// Mitsubishi GX Works2 project: test1   PLC: Q03UDV

PROGRAM MAIN
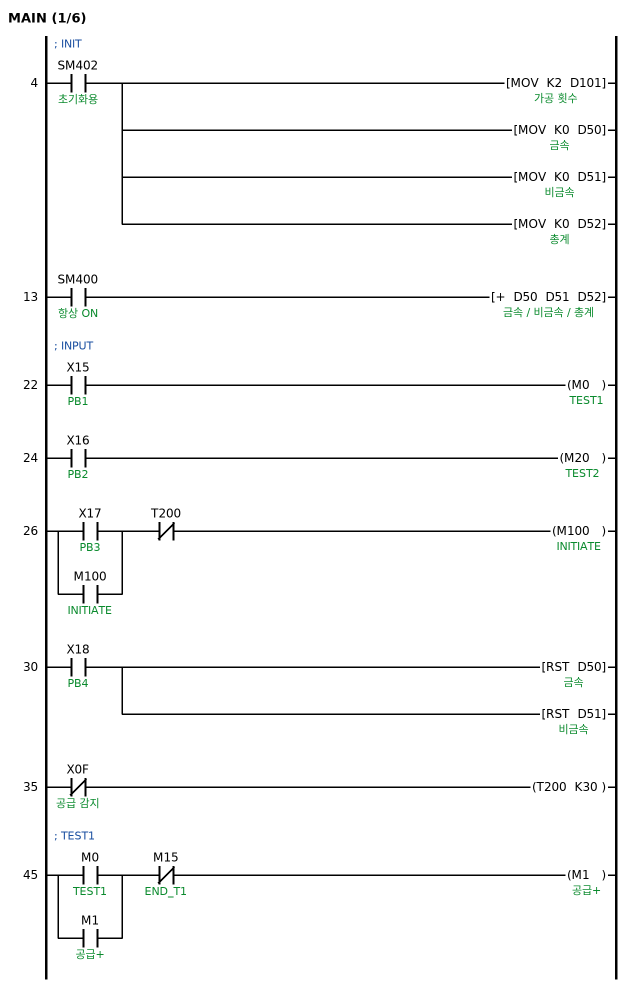
; INIT
4     LD      SM402  ; 초기화용
      MOV     K2 D101  ; 가공 횟수
      MOV     K0 D50  ; 금속
      MOV     K0 D51  ; 비금속
      MOV     K0 D52  ; 총계
13    LD      SM400  ; 항상 ON
      +       D50 D51 D52
; INPUT
22    LD      X15  ; PB1
      OUT     M0  ; TEST1
24    LD      X16  ; PB2
      OUT     M20  ; TEST2
26    LD      X17  ; PB3
      OR      M100  ; INITIATE
      ANI     T200
      OUT     M100  ; INITIATE
30    LD      X18  ; PB4
      RST     D50  ; 금속
      RST     D51  ; 비금속
35    LDI     X0F  ; 공급 감지
      OUT     T200 K30
; TEST1
45    LD      M0  ; TEST1
      OR      M1  ; 공급+
      ANI     M15  ; END_T1
      OUT     M1  ; 공급+
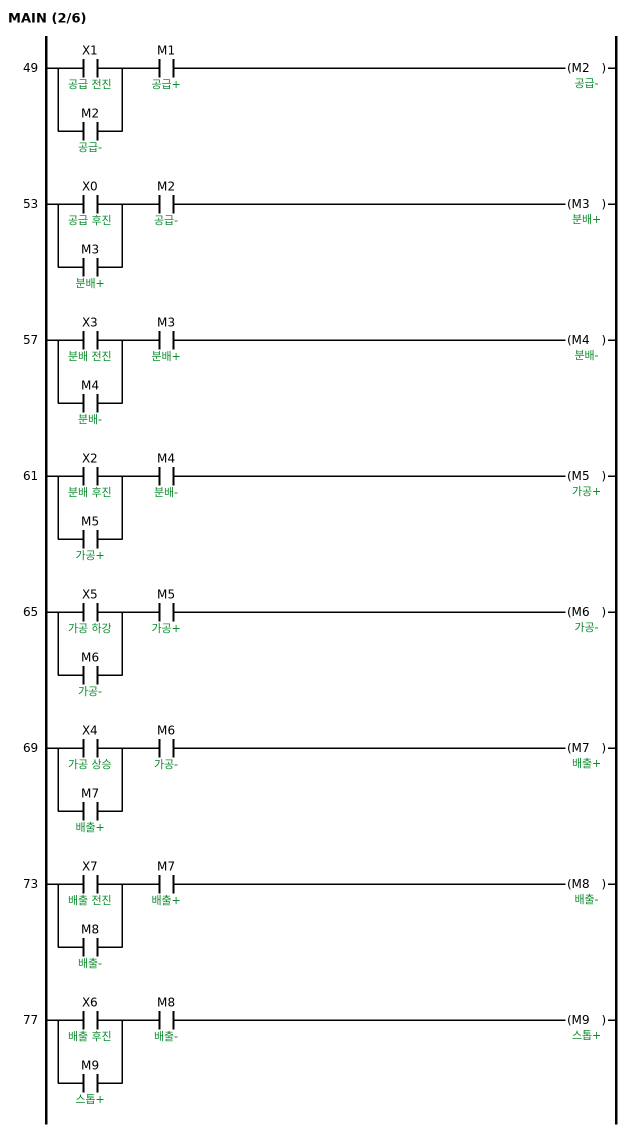
49    LD      X1  ; 공급 전진
      OR      M2  ; 공급-
      AND     M1  ; 공급+
      OUT     M2  ; 공급-
53    LD      X0  ; 공급 후진
      OR      M3  ; 분배+
      AND     M2  ; 공급-
      OUT     M3  ; 분배+
57    LD      X3  ; 분배 전진
      OR      M4  ; 분배-
      AND     M3  ; 분배+
      OUT     M4  ; 분배-
61    LD      X2  ; 분배 후진
      OR      M5  ; 가공+
      AND     M4  ; 분배-
      OUT     M5  ; 가공+
65    LD      X5  ; 가공 하강
      OR      M6  ; 가공-
      AND     M5  ; 가공+
      OUT     M6  ; 가공-
69    LD      X4  ; 가공 상승
      OR      M7  ; 배출+
      AND     M6  ; 가공-
      OUT     M7  ; 배출+
73    LD      X7  ; 배출 전진
      OR      M8  ; 배출-
      AND     M7  ; 배출+
      OUT     M8  ; 배출-
77    LD      X6  ; 배출 후진
      OR      M9  ; 스톱+
      AND     M8  ; 배출-
      OUT     M9  ; 스톱+
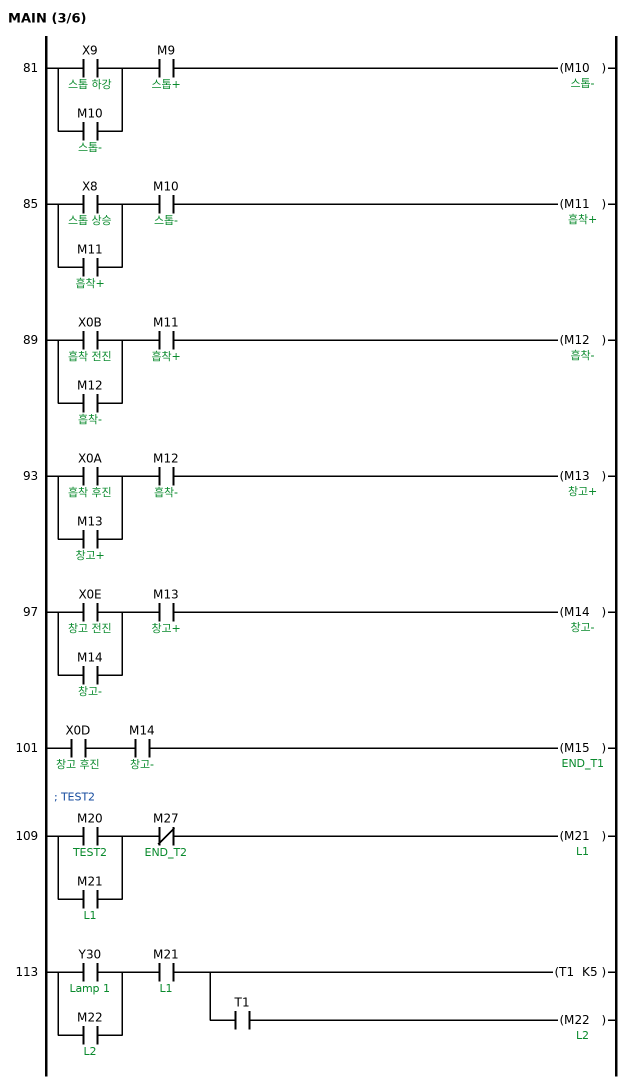
81    LD      X9  ; 스톱 하강
      OR      M10  ; 스톱-
      AND     M9  ; 스톱+
      OUT     M10  ; 스톱-
85    LD      X8  ; 스톱 상승
      OR      M11  ; 흡착+
      AND     M10  ; 스톱-
      OUT     M11  ; 흡착+
89    LD      X0B  ; 흡착 전진
      OR      M12  ; 흡착-
      AND     M11  ; 흡착+
      OUT     M12  ; 흡착-
93    LD      X0A  ; 흡착 후진
      OR      M13  ; 창고+
      AND     M12  ; 흡착-
      OUT     M13  ; 창고+
97    LD      X0E  ; 창고 전진
      OR      M14  ; 창고-
      AND     M13  ; 창고+
      OUT     M14  ; 창고-
101   LD      X0D  ; 창고 후진
      AND     M14  ; 창고-
      OUT     M15  ; END_T1
; TEST2
109   LD      M20  ; TEST2
      OR      M21  ; L1
      ANI     M27  ; END_T2
      OUT     M21  ; L1
113   LD      Y30  ; Lamp 1
      OR      M22  ; L2
      AND     M21  ; L1
      OUT     T1 K5
      AND     T1
      OUT     M22  ; L2
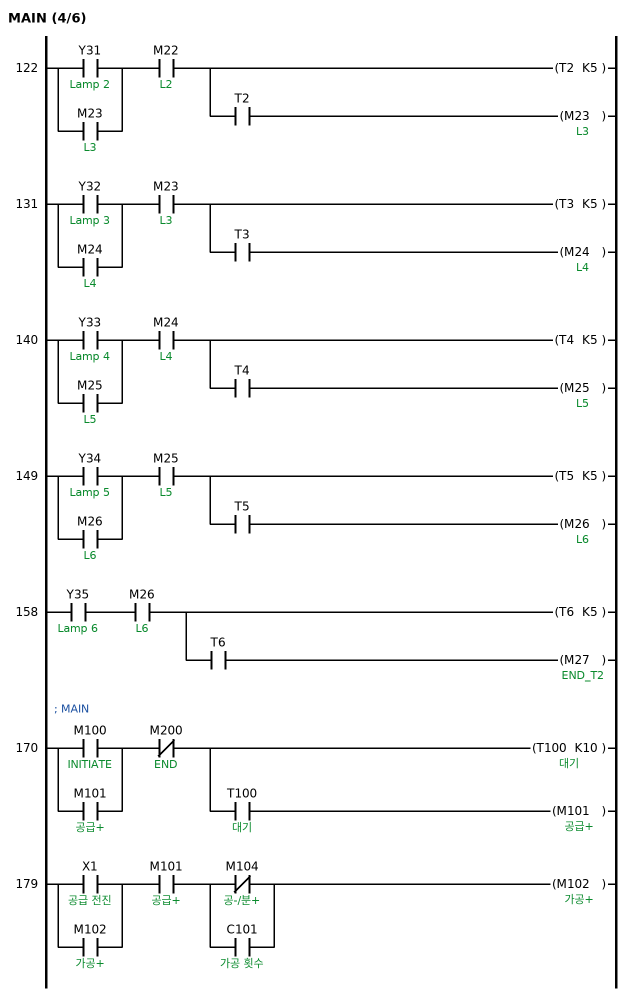
122   LD      Y31  ; Lamp 2
      OR      M23  ; L3
      AND     M22  ; L2
      OUT     T2 K5
      AND     T2
      OUT     M23  ; L3
131   LD      Y32  ; Lamp 3
      OR      M24  ; L4
      AND     M23  ; L3
      OUT     T3 K5
      AND     T3
      OUT     M24  ; L4
140   LD      Y33  ; Lamp 4
      OR      M25  ; L5
      AND     M24  ; L4
      OUT     T4 K5
      AND     T4
      OUT     M25  ; L5
149   LD      Y34  ; Lamp 5
      OR      M26  ; L6
      AND     M25  ; L5
      OUT     T5 K5
      AND     T5
      OUT     M26  ; L6
158   LD      Y35  ; Lamp 6
      AND     M26  ; L6
      OUT     T6 K5
      AND     T6
      OUT     M27  ; END_T2
; MAIN
170   LD      M100  ; INITIATE
      OR      M101  ; 공급+
      ANI     M200  ; END
      OUT     T100 K10  ; 대기
      AND     T100  ; 대기
      OUT     M101  ; 공급+
179   LD      X1  ; 공급 전진
      OR      M102  ; 가공+
      AND     M101  ; 공급+
      LDI     M104  ; 공-/분+
      OR      C101  ; 가공 횟수
      ANB
      OUT     M102  ; 가공+
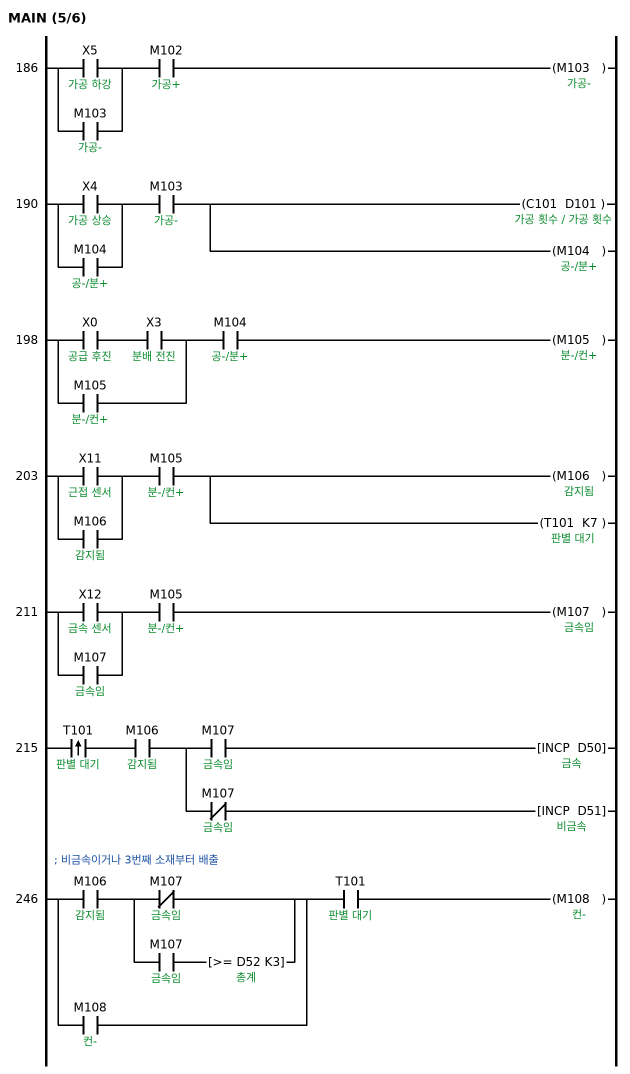
186   LD      X5  ; 가공 하강
      OR      M103  ; 가공-
      AND     M102  ; 가공+
      OUT     M103  ; 가공-
190   LD      X4  ; 가공 상승
      OR      M104  ; 공-/분+
      AND     M103  ; 가공-
      OUT     C101 D101  ; 가공 횟수 / 가공 횟수
      OUT     M104  ; 공-/분+
198   LD      X0  ; 공급 후진
      AND     X3  ; 분배 전진
      OR      M105  ; 분-/컨+
      AND     M104  ; 공-/분+
      OUT     M105  ; 분-/컨+
203   LD      X11  ; 근접 센서
      OR      M106  ; 감지됨
      AND     M105  ; 분-/컨+
      OUT     M106  ; 감지됨
      OUT     T101 K7  ; 판별 대기
211   LD      X12  ; 금속 센서
      OR      M107  ; 금속임
      AND     M105  ; 분-/컨+
      OUT     M107  ; 금속임
215   LDP     T101  ; 판별 대기
      AND     M106  ; 감지됨
      MPS
      AND     M107  ; 금속임
      INCP    D50
      MPP
      ANI     M107  ; 금속임
      INCP    D51
; 비금속이거나 3번째 소재부터 배출
246   LD      M106  ; 감지됨
      LDI     M107  ; 금속임
      LD      M107  ; 금속임
      AND>=   D52 K3  ; 총계
      ORB
      ANB
      OR      M108  ; 컨-
      AND     T101  ; 판별 대기
      OUT     M108  ; 컨-
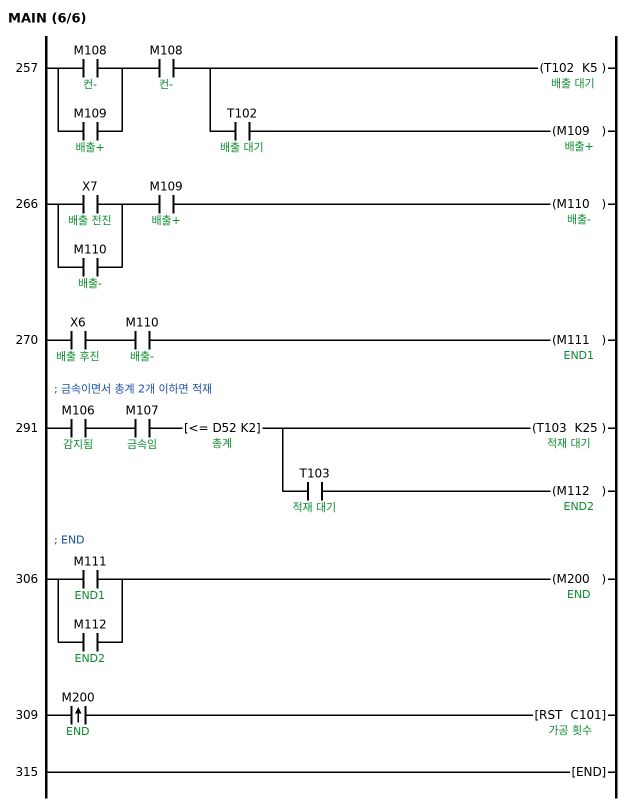
257   LD      M108  ; 컨-
      OR      M109  ; 배출+
      AND     M108  ; 컨-
      OUT     T102 K5  ; 배출 대기
      AND     T102  ; 배출 대기
      OUT     M109  ; 배출+
266   LD      X7  ; 배출 전진
      OR      M110  ; 배출-
      AND     M109  ; 배출+
      OUT     M110  ; 배출-
270   LD      X6  ; 배출 후진
      AND     M110  ; 배출-
      OUT     M111  ; END1
; 금속이면서 총계 2개 이하면 적재
291   LD      M106  ; 감지됨
      AND     M107  ; 금속임
      AND<=   D52 K2  ; 총계
      OUT     T103 K25  ; 적재 대기
      AND     T103  ; 적재 대기
      OUT     M112  ; END2
; END
306   LD      M111  ; END1
      OR      M112  ; END2
      OUT     M200  ; END
309   LDP     M200  ; END
      RST     C101  ; 가공 횟수
315   END
END_PROGRAM

PROGRAM OUTPUT
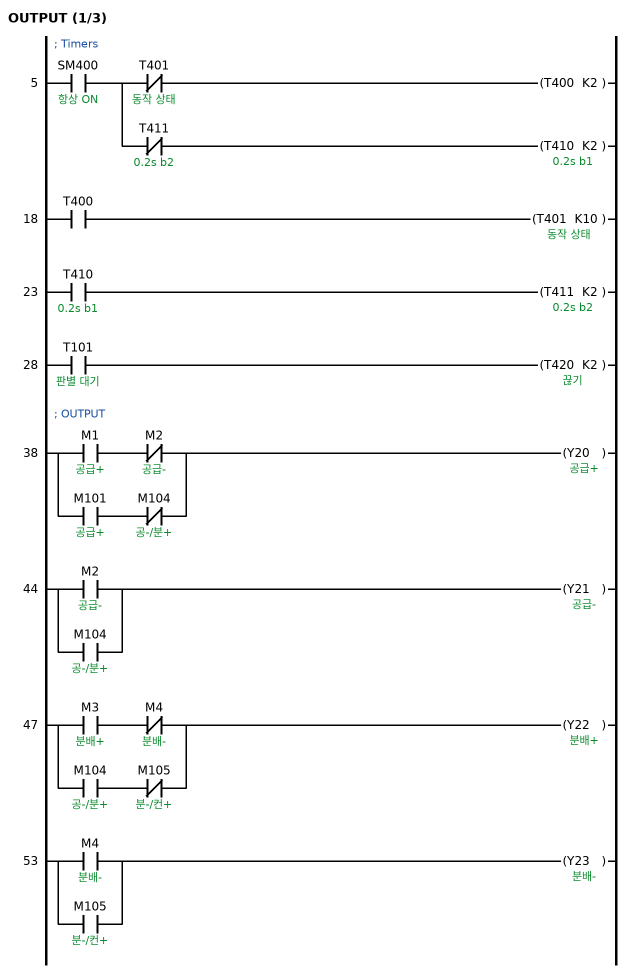
; Timers
5     LD      SM400  ; 항상 ON
      MPS
      ANI     T401  ; 동작 상태
      OUT     T400 K2
      MPP
      ANI     T411  ; 0.2s b2
      OUT     T410 K2  ; 0.2s b1
18    LD      T400
      OUT     T401 K10  ; 동작 상태
23    LD      T410  ; 0.2s b1
      OUT     T411 K2  ; 0.2s b2
28    LD      T101  ; 판별 대기
      OUT     T420 K2  ; 끊기
; OUTPUT
38    LD      M1  ; 공급+
      ANI     M2  ; 공급-
      LD      M101  ; 공급+
      ANI     M104  ; 공-/분+
      ORB
      OUT     Y20  ; 공급+
44    LD      M2  ; 공급-
      OR      M104  ; 공-/분+
      OUT     Y21  ; 공급-
47    LD      M3  ; 분배+
      ANI     M4  ; 분배-
      LD      M104  ; 공-/분+
      ANI     M105  ; 분-/컨+
      ORB
      OUT     Y22  ; 분배+
53    LD      M4  ; 분배-
      OR      M105  ; 분-/컨+
      OUT     Y23  ; 분배-
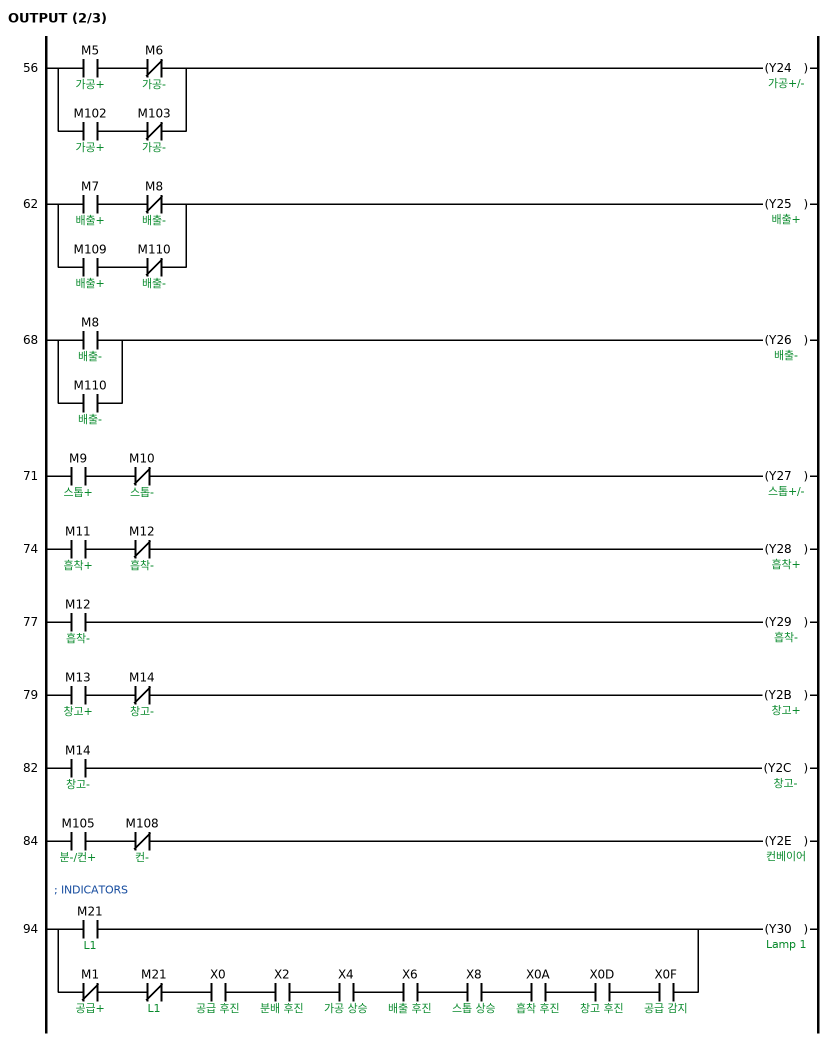
56    LD      M5  ; 가공+
      ANI     M6  ; 가공-
      LD      M102  ; 가공+
      ANI     M103  ; 가공-
      ORB
      OUT     Y24  ; 가공+/-
62    LD      M7  ; 배출+
      ANI     M8  ; 배출-
      LD      M109  ; 배출+
      ANI     M110  ; 배출-
      ORB
      OUT     Y25  ; 배출+
68    LD      M8  ; 배출-
      OR      M110  ; 배출-
      OUT     Y26  ; 배출-
71    LD      M9  ; 스톱+
      ANI     M10  ; 스톱-
      OUT     Y27  ; 스톱+/-
74    LD      M11  ; 흡착+
      ANI     M12  ; 흡착-
      OUT     Y28  ; 흡착+
77    LD      M12  ; 흡착-
      OUT     Y29  ; 흡착-
79    LD      M13  ; 창고+
      ANI     M14  ; 창고-
      OUT     Y2B  ; 창고+
82    LD      M14  ; 창고-
      OUT     Y2C  ; 창고-
84    LD      M105  ; 분-/컨+
      ANI     M108  ; 컨-
      OUT     Y2E  ; 컨베이어
; INDICATORS
94    LD      M21  ; L1
      LDI     M1  ; 공급+
      ANI     M21  ; L1
      AND     X0  ; 공급 후진
      AND     X2  ; 분배 후진
      AND     X4  ; 가공 상승
      AND     X6  ; 배출 후진
      AND     X8  ; 스톱 상승
      AND     X0A  ; 흡착 후진
      AND     X0D  ; 창고 후진
      AND     X0F  ; 공급 감지
      ORB
      OUT     Y30  ; Lamp 1
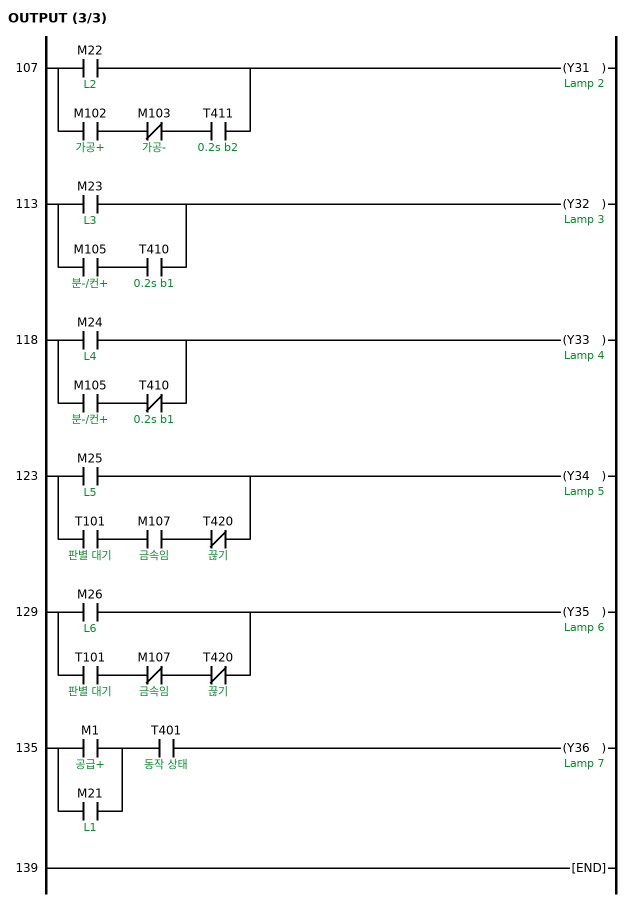
107   LD      M22  ; L2
      LD      M102  ; 가공+
      ANI     M103  ; 가공-
      AND     T411  ; 0.2s b2
      ORB
      OUT     Y31  ; Lamp 2
113   LD      M23  ; L3
      LD      M105  ; 분-/컨+
      AND     T410  ; 0.2s b1
      ORB
      OUT     Y32  ; Lamp 3
118   LD      M24  ; L4
      LD      M105  ; 분-/컨+
      ANI     T410  ; 0.2s b1
      ORB
      OUT     Y33  ; Lamp 4
123   LD      M25  ; L5
      LD      T101  ; 판별 대기
      AND     M107  ; 금속임
      ANI     T420  ; 끊기
      ORB
      OUT     Y34  ; Lamp 5
129   LD      M26  ; L6
      LD      T101  ; 판별 대기
      ANI     M107  ; 금속임
      ANI     T420  ; 끊기
      ORB
      OUT     Y35  ; Lamp 6
135   LD      M1  ; 공급+
      OR      M21  ; L1
      AND     T401  ; 동작 상태
      OUT     Y36  ; Lamp 7
139   END
END_PROGRAM
